(* CODESYS project xlh_gantry_00_04.project
   Description: Receives some incoming messages and echoes them with CAN-ID +1
   Company: 3S - Smart Software Solutions GmbH
   Version: 1.0.0.0
   Title: CAN Bus API Example
   Author: 3S - Smart Software Solutions GmbH

Project tree, tasks and I/O mapping:
  xLH_base : CODESYS Control for Raspberry Pi 64 SL, CODESYS, order no. 2302000009, version 4.20.0.0
    application app
      libraries: Standard, 3.5.22.0 (System); Util, 3.5.22.0 (System); VisuDialogs, * (System); Memory, * (3S - Smart Software Solutions GmbH); CmpBitmapPool, * (System); CAN API, 1.0.0.4 (CODESYS); MemoryUtils, * (3S - Smart Software Solutions GmbH); CAA CiA 405, 4.3.0.0 (CODESYS)
      task CANOPEN_TASK (cyclic, interval 1 ms, priority 1) calls nothing
      task VISU_TASK (cyclic, interval 100 ms, priority 31) calls VisuElems.Visu_Prg
      task MAIN_TASK (cyclic, interval 4 ms, priority 2) calls io, MAIN_CALLER
      task SoftMotion_PlanningTask (cyclic, interval t#2ms, priority 15) calls nothing
      program MAIN_CALLER [ST]
      trace Trace_AxX (task MAIN_TASK): x_axis.fActPosition, x_axis.fSetPosition, x_axis.fSetAcceleration, x_axis.fActAcceleration, x_axis.fSetVelocity, x_axis.fActVelocity, io.motion.adiFrequency[1]
      visualisation Visualization
      trace Trace (task MAIN_TASK): MC.diPosition, MC.iSetSpeed, MC.iDebug2Pos, MC.iDebug1Mileage, MC.auiUltrasonic[1], MC.fbReadStatusLoopTime.udiValue, MC.iSpeed2, MC.iSpeed1, MC.iPitch
      data type MOTION_CONTROL_BYTE
      MOTION_BASE/
        function block FB_XLH_MOTION_AXIS_SIMPLE_ES [ST]: mRead
        function block FB_PLC_OPEN_AXIS [ST]: plcOpen, executeToFalse
        function block FB_XLH_MOTION_AXIS_SIMPLE [ST]
        function block FB_XLH_MOTION_AXIS_BASE [ST]: mRead, mWrite
        function block FB_AXG_MOVE_ABSOLUTE [ST]
        function block FB_AXG_MOVE_RELATIVE [ST]
        function block FB_AXG_PICK_AND_PLACE [ST]
        function block FB_KALMAN_FILTER [ST]: reset
      IO/
        function block FB_XLH_MOTION [ST]: read, write
        program io [ST]: read, write
        function block FB_XLH_GPIO [ST]: read, write
        function block FB_XLH_DXL_RGB [ST]: read, write
      program MC [ST]: write, read, axSmExecuteToFalse, axGexecuteToFalse
      axis group AxisGroup: TRAFO.Kin_Gantry3, axes x_axis, y_axis, z_axis
      trace Trace_AxZ (task MAIN_TASK): z_axis.fActPosition, z_axis.fSetPosition, z_axis.fSetAcceleration, z_axis.fActAcceleration, z_axis.fSetVelocity, z_axis.fActVelocity, io.motion.adiFrequency[3]
    CANbus : CANbus, CODESYS, version 4.3.0.0
        settings: Baudrate = 1000 kbit/s
      CANopen_Manager : CANopen_Manager, CODESYS, version 4.3.0.0
          settings: NMT Start All = TRUE; Polling of optional slaves = FALSE; ConfigVersion = 50659584
        xlh_dynamixel_rgb : xlh_stamp_dynamixel_rgb, xemax ag, order no. 0, version Revision=16#00000001, FileVersion=1.0 (disabled)
            settings: NODEIDSAVED = 2; SDO Timeout = 1000000; PDO_Autoconfig = FALSE; EXPERTSETTINGS = FALSE; PDO 16#1400.COBID = 16#00000202; Process by CANopenManager = TRUE; PDO 16#1401.COBID = 16#00000302; Process by CANopenManager = TRUE; PDO 16#1402.COBID = 16#00000402; Process by CANopenManager = TRUE; PDO 16#1800.COBID = 16#00000182; Process by CANopenManager = TRUE; Dxl 1 Control.Subindex = 16#01; Dxl 1 Position.Subindex = 16#02; Dxl 1 Velocity.Subindex = 16#03; Dxl 2 Control.Subindex = 16#04; Dxl 2 Position.Subindex = 16#05; Dxl 2 Velocity.Subindex = 16#06; RGB red.Subindex = 16#01; RGB green.Subindex = 16#02; RGB blue.Subindex = 16#03; Dxl 1  Position read.Subindex = 16#01; Dxl 1 Current read.Subindex = 16#02; Dxl 2  Position read.Subindex = 16#03; Dxl 2 Current read.Subindex = 16#04; SDO List.Set COB-ID sync.Index = 16#1005; SDO List.Set COB-ID sync.Subindex = 16#00; SDO List.Set COB-ID sync.Value = 16#00000080; SDO List.Set COB-ID sync.Size = 32; SDO List.Set COB-ID sync.AbortIfError = FALSE; SDO List.Set COB-ID sync.JumpToLine = FALSE; SDO List.Set COB-ID sync.Line = 0; SDO List.Set communication cycle period.Index = 16#1006; SDO List.Set communication cycle period.Subindex = 16#00; SDO List.Set communication cycle period.Value = 16#00000000; SDO List.Set communication cycle period.Size = 32; SDO List.Set communication cycle period.AbortIfError = FALSE; SDO List.Set communication cycle period.JumpToLine = FALSE; SDO List.Set communication cycle period.Line = 0; SDO List.Set Guardtime.Index = 16#100C;
              SDO List.Set Guardtime.Subindex = 16#00; SDO List.Set Guardtime.Value = 16#000000C8; SDO List.Set Guardtime.Size = 16; SDO List.Set Guardtime.AbortIfError = FALSE; SDO List.Set Guardtime.JumpToLine = FALSE; SDO List.Set Guardtime.Line = 0; SDO List.Set Lifetime.Index = 16#100D; SDO List.Set Lifetime.Subindex = 16#00; SDO List.Set Lifetime.Value = 16#00000003; SDO List.Set Lifetime.Size = 8; SDO List.Set Lifetime.AbortIfError = FALSE; SDO List.Set Lifetime.JumpToLine = FALSE; SDO List.Set Lifetime.Line = 0; SDO List.Set Heartbeat Consumer.Index = 16#1016; SDO List.Set Heartbeat Consumer.Subindex = 16#01; SDO List.Set Heartbeat Consumer.Value = 0; SDO List.Set Heartbeat Consumer.Size = 32; SDO List.Set Heartbeat Consumer.AbortIfError = FALSE; SDO List.Set Heartbeat Consumer.JumpToLine = FALSE; SDO List.Set Heartbeat Consumer.Line = 0; SDO List.Disable PDO.Index = 16#1400; SDO List.Disable PDO.Subindex = 16#01; SDO List.Disable PDO.Value = 16#80000202; SDO List.Disable PDO.Size = 32; SDO List.Disable PDO.AbortIfError = FALSE; SDO List.Disable PDO.JumpToLine = FALSE; SDO List.Disable PDO.Line = 0; SDO List.Set transmission type.Index = 16#1400; SDO List.Set transmission type.Subindex = 16#02; SDO List.Set transmission type.Value = 16#FF; SDO List.Set transmission type.Size = 8; SDO List.Set transmission type.AbortIfError = FALSE; SDO List.Set transmission type.JumpToLine = FALSE; SDO List.Set transmission type.Line = 0; SDO List.Set and enable COB-ID.Index = 16#1400; SDO List.Set and enable COB-ID.Subindex = 16#01; SDO List.Set and enable COB-ID.Value = 16#00000202; SDO List.Set and enable COB-ID.Size = 32; SDO List.Set and enable COB-ID.AbortIfError = FALSE; SDO List.Set and enable COB-ID.JumpToLine = FALSE;
              SDO List.Set and enable COB-ID.Line = 0; SDO List.Disable PDO.Index = 16#1401; SDO List.Disable PDO.Subindex = 16#01; SDO List.Disable PDO.Value = 16#80000302; SDO List.Disable PDO.Size = 32; SDO List.Disable PDO.AbortIfError = FALSE; SDO List.Disable PDO.JumpToLine = FALSE; SDO List.Disable PDO.Line = 0; SDO List.Set transmission type.Index = 16#1401; SDO List.Set transmission type.Subindex = 16#02; SDO List.Set transmission type.Value = 16#FF; SDO List.Set transmission type.Size = 8; SDO List.Set transmission type.AbortIfError = FALSE; SDO List.Set transmission type.JumpToLine = FALSE; SDO List.Set transmission type.Line = 0; SDO List.Set and enable COB-ID.Index = 16#1401; SDO List.Set and enable COB-ID.Subindex = 16#01; SDO List.Set and enable COB-ID.Value = 16#00000302; SDO List.Set and enable COB-ID.Size = 32; SDO List.Set and enable COB-ID.AbortIfError = FALSE; SDO List.Set and enable COB-ID.JumpToLine = FALSE; SDO List.Set and enable COB-ID.Line = 0; SDO List.Disable PDO.Index = 16#1402; SDO List.Disable PDO.Subindex = 16#01; SDO List.Disable PDO.Value = 16#80000402; SDO List.Disable PDO.Size = 32; SDO List.Disable PDO.AbortIfError = FALSE; SDO List.Disable PDO.JumpToLine = FALSE; SDO List.Disable PDO.Line = 0; SDO List.Set transmission type.Index = 16#1402; SDO List.Set transmission type.Subindex = 16#02; SDO List.Set transmission type.Value = 16#FF; SDO List.Set transmission type.Size = 8; SDO List.Set transmission type.AbortIfError = FALSE; SDO List.Set transmission type.JumpToLine = FALSE; SDO List.Set transmission type.Line = 0; SDO List.Set and enable COB-ID.Index = 16#1402; SDO List.Set and enable COB-ID.Subindex = 16#01; SDO List.Set and enable COB-ID.Value = 16#00000402; SDO List.Set and enable COB-ID.Size = 32;
              SDO List.Set and enable COB-ID.AbortIfError = FALSE; SDO List.Set and enable COB-ID.JumpToLine = FALSE; SDO List.Set and enable COB-ID.Line = 0; SDO List.Disable PDO.Index = 16#1800; SDO List.Disable PDO.Subindex = 16#01; SDO List.Disable PDO.Value = 16#80000182; SDO List.Disable PDO.Size = 32; SDO List.Disable PDO.AbortIfError = FALSE; SDO List.Disable PDO.JumpToLine = FALSE; SDO List.Disable PDO.Line = 0; SDO List.Set transmission type.Index = 16#1800; SDO List.Set transmission type.Subindex = 16#02; SDO List.Set transmission type.Value = 16#FF; SDO List.Set transmission type.Size = 8; SDO List.Set transmission type.AbortIfError = FALSE; SDO List.Set transmission type.JumpToLine = FALSE; SDO List.Set transmission type.Line = 0; SDO List.Set inhibit time.Index = 16#1800; SDO List.Set inhibit time.Subindex = 16#03; SDO List.Set inhibit time.Value = 16#0000; SDO List.Set inhibit time.Size = 16; SDO List.Set inhibit time.AbortIfError = FALSE; SDO List.Set inhibit time.JumpToLine = FALSE; SDO List.Set inhibit time.Line = 0; SDO List.Set event time.Index = 16#1800; SDO List.Set event time.Subindex = 16#05; SDO List.Set event time.Value = 16#0000; SDO List.Set event time.Size = 16; SDO List.Set event time.AbortIfError = FALSE; SDO List.Set event time.JumpToLine = FALSE; SDO List.Set event time.Line = 0; SDO List.Set and enable COB-ID.Index = 16#1800; SDO List.Set and enable COB-ID.Subindex = 16#01; SDO List.Set and enable COB-ID.Value = 16#00000182; SDO List.Set and enable COB-ID.Size = 32; SDO List.Set and enable COB-ID.AbortIfError = FALSE; SDO List.Set and enable COB-ID.JumpToLine = FALSE; SDO List.Set and enable COB-ID.Line = 0; ConfigVersion = 50659584
            output app.io.dxlRgb.bDxl1Torque : BOOL  // Dxl 1 Control.Bit0
            output app.io.dxlRgb.bDxl1Led : BOOL  // Dxl 1 Control.Bit1
            output app.io.dxlRgb.uiDxl1Position : UINT  // Dxl 1 Position
            output app.io.dxlRgb.uiDxl1Velocity : UINT  // Dxl 1 Velocity
            output app.io.dxlRgb.bDxl2Torque : BOOL  // Dxl 2 Control.Bit0
            output app.io.dxlRgb.bDxl2Led : BOOL  // Dxl 2 Control.Bit1
            output app.io.dxlRgb.uiDxl2Position : UINT  // Dxl 2 Position
            output app.io.dxlRgb.uiDxl2Velocity : UINT  // Dxl 2 Velocity
            output app.io.dxlRgb.byRgbRed : USINT  // RGB red
            output app.io.dxlRgb.byRgbGreen : USINT  // RGB green
            output app.io.dxlRgb.byRgbBlue : USINT  // RGB blue
            input  app.io.dxlRgb.uiDxl1PositionGet : UINT  // Dxl 1  Position read
            input  app.io.dxlRgb.iDxl1CurrentGet : INT  // Dxl 1 Current read
            input  app.io.dxlRgb.uiDxl2PositionGet : UINT  // Dxl 2  Position read
            input  app.io.dxlRgb.iDxl2CurrentGet : INT  // Dxl 2 Current read
            unmapped channels: Dxl 1 Control, Dxl 2 Control
        xlh_motion : xlh_motion, xemax ag, order no. 0, version Revision=16#00000001, FileVersion=1.0
            settings: NODEIDSAVED = 1; SDO Timeout = 1000000; PDO_Autoconfig = FALSE; EXPERTSETTINGS = True; PDO 16#1400.COBID = 16#00000201; Process by CANopenManager = TRUE; PDO 16#1401.COBID = 16#00000301; Process by CANopenManager = TRUE; PDO 16#1402.COBID = 16#00000401; Process by CANopenManager = TRUE; PDO 16#1403.COBID = 16#00000501; Process by CANopenManager = TRUE; PDO 16#1800.COBID = 16#00000181; Process by CANopenManager = TRUE; PDO 16#1801.COBID = 16#00000281; Process by CANopenManager = TRUE; PDO 16#1802.COBID = 16#00000381; Process by CANopenManager = TRUE; Control 1.Subindex = 16#01; Control 2.Subindex = 16#02; Control 3.Subindex = 16#03; Control 4.Subindex = 16#04; Outputs 0-7.Subindex = 16#01; Outputs 8-15.Subindex = 16#02; Magnet Duty Cycle.Subindex = 16#01; Freqeuncy 1.Subindex = 16#05; Freqeuncy 2.Subindex = 16#06; Freqeuncy 3.Subindex = 16#07; Freqeuncy 4.Subindex = 16#08; Servo 1.Subindex = 16#01; Servo 2.Subindex = 16#02; Servo 3.Subindex = 16#03; Servo 4.Subindex = 16#04; Servo 5.Subindex = 16#05; Servo 6.Subindex = 16#06; Servo 7.Subindex = 16#07; Servo 8.Subindex = 16#08; Position 1.Subindex = 16#01; Position 2.Subindex = 16#02; Position 3.Subindex = 16#03;
              Position 4.Subindex = 16#04; Inputs 0-7.Subindex = 16#01; Inputs 8-15.Subindex = 16#02; Inputs CLK.Subindex = 16#03; SDO List.Set COB-ID sync.Index = 16#1005; SDO List.Set COB-ID sync.Subindex = 16#00; SDO List.Set COB-ID sync.Value = 16#00000080; SDO List.Set COB-ID sync.Size = 32; SDO List.Set COB-ID sync.AbortIfError = FALSE; SDO List.Set COB-ID sync.JumpToLine = FALSE; SDO List.Set COB-ID sync.Line = 0; SDO List.Set communication cycle period.Index = 16#1006; SDO List.Set communication cycle period.Subindex = 16#00; SDO List.Set communication cycle period.Value = 16#00000000; SDO List.Set communication cycle period.Size = 32; SDO List.Set communication cycle period.AbortIfError = FALSE; SDO List.Set communication cycle period.JumpToLine = FALSE; SDO List.Set communication cycle period.Line = 0; SDO List.Set Guardtime.Index = 16#100C; SDO List.Set Guardtime.Subindex = 16#00; SDO List.Set Guardtime.Value = 16#000000C8; SDO List.Set Guardtime.Size = 16; SDO List.Set Guardtime.AbortIfError = FALSE; SDO List.Set Guardtime.JumpToLine = FALSE; SDO List.Set Guardtime.Line = 0; SDO List.Set Lifetime.Index = 16#100D; SDO List.Set Lifetime.Subindex = 16#00; SDO List.Set Lifetime.Value = 16#00000003; SDO List.Set Lifetime.Size = 8; SDO List.Set Lifetime.AbortIfError = FALSE; SDO List.Set Lifetime.JumpToLine = FALSE; SDO List.Set Lifetime.Line = 0; SDO List.Set Heartbeat Consumer.Index = 16#1016; SDO List.Set Heartbeat Consumer.Subindex = 16#01; SDO List.Set Heartbeat Consumer.Value = 0; SDO List.Set Heartbeat Consumer.Size = 32; SDO List.Set Heartbeat Consumer.AbortIfError = FALSE; SDO List.Set Heartbeat Consumer.JumpToLine = FALSE; SDO List.Set Heartbeat Consumer.Line = 0; SDO List.Disable PDO.Index = 16#1400;
              SDO List.Disable PDO.Subindex = 16#01; SDO List.Disable PDO.Value = 16#80000201; SDO List.Disable PDO.Size = 32; SDO List.Disable PDO.AbortIfError = FALSE; SDO List.Disable PDO.JumpToLine = FALSE; SDO List.Disable PDO.Line = 0; SDO List.Set transmission type.Index = 16#1400; SDO List.Set transmission type.Subindex = 16#02; SDO List.Set transmission type.Value = 16#FF; SDO List.Set transmission type.Size = 8; SDO List.Set transmission type.AbortIfError = FALSE; SDO List.Set transmission type.JumpToLine = FALSE; SDO List.Set transmission type.Line = 0; SDO List.Set and enable COB-ID.Index = 16#1400; SDO List.Set and enable COB-ID.Subindex = 16#01; SDO List.Set and enable COB-ID.Value = 16#00000201; SDO List.Set and enable COB-ID.Size = 32; SDO List.Set and enable COB-ID.AbortIfError = FALSE; SDO List.Set and enable COB-ID.JumpToLine = FALSE; SDO List.Set and enable COB-ID.Line = 0; SDO List.Disable PDO.Index = 16#1401; SDO List.Disable PDO.Subindex = 16#01; SDO List.Disable PDO.Value = 16#80000301; SDO List.Disable PDO.Size = 32; SDO List.Disable PDO.AbortIfError = FALSE; SDO List.Disable PDO.JumpToLine = FALSE; SDO List.Disable PDO.Line = 0; SDO List.Set transmission type.Index = 16#1401; SDO List.Set transmission type.Subindex = 16#02; SDO List.Set transmission type.Value = 16#FF; SDO List.Set transmission type.Size = 8; SDO List.Set transmission type.AbortIfError = FALSE; SDO List.Set transmission type.JumpToLine = FALSE; SDO List.Set transmission type.Line = 0; SDO List.Set and enable COB-ID.Index = 16#1401; SDO List.Set and enable COB-ID.Subindex = 16#01; SDO List.Set and enable COB-ID.Value = 16#00000301; SDO List.Set and enable COB-ID.Size = 32; SDO List.Set and enable COB-ID.AbortIfError = FALSE; SDO List.Set and enable COB-ID.JumpToLine = FALSE;
              SDO List.Set and enable COB-ID.Line = 0; SDO List.Disable PDO.Index = 16#1402; SDO List.Disable PDO.Subindex = 16#01; SDO List.Disable PDO.Value = 16#80000401; SDO List.Disable PDO.Size = 32; SDO List.Disable PDO.AbortIfError = FALSE; SDO List.Disable PDO.JumpToLine = FALSE; SDO List.Disable PDO.Line = 0; SDO List.Set transmission type.Index = 16#1402; SDO List.Set transmission type.Subindex = 16#02; SDO List.Set transmission type.Value = 16#FF; SDO List.Set transmission type.Size = 8; SDO List.Set transmission type.AbortIfError = FALSE; SDO List.Set transmission type.JumpToLine = FALSE; SDO List.Set transmission type.Line = 0; SDO List.Set and enable COB-ID.Index = 16#1402; SDO List.Set and enable COB-ID.Subindex = 16#01; SDO List.Set and enable COB-ID.Value = 16#00000401; SDO List.Set and enable COB-ID.Size = 32; SDO List.Set and enable COB-ID.AbortIfError = FALSE; SDO List.Set and enable COB-ID.JumpToLine = FALSE; SDO List.Set and enable COB-ID.Line = 0; SDO List.Disable PDO.Index = 16#1403; SDO List.Disable PDO.Subindex = 16#01; SDO List.Disable PDO.Value = 16#80000501; SDO List.Disable PDO.Size = 32; SDO List.Disable PDO.AbortIfError = FALSE; SDO List.Disable PDO.JumpToLine = FALSE; SDO List.Disable PDO.Line = 0; SDO List.Set transmission type.Index = 16#1403; SDO List.Set transmission type.Subindex = 16#02; SDO List.Set transmission type.Value = 16#FF; SDO List.Set transmission type.Size = 8; SDO List.Set transmission type.AbortIfError = FALSE; SDO List.Set transmission type.JumpToLine = FALSE; SDO List.Set transmission type.Line = 0; SDO List.Set and enable COB-ID.Index = 16#1403; SDO List.Set and enable COB-ID.Subindex = 16#01; SDO List.Set and enable COB-ID.Value = 16#00000501; SDO List.Set and enable COB-ID.Size = 32;
              SDO List.Set and enable COB-ID.AbortIfError = FALSE; SDO List.Set and enable COB-ID.JumpToLine = FALSE; SDO List.Set and enable COB-ID.Line = 0; SDO List.Disable PDO.Index = 16#1800; SDO List.Disable PDO.Subindex = 16#01; SDO List.Disable PDO.Value = 16#80000181; SDO List.Disable PDO.Size = 32; SDO List.Disable PDO.AbortIfError = FALSE; SDO List.Disable PDO.JumpToLine = FALSE; SDO List.Disable PDO.Line = 0; SDO List.Set transmission type.Index = 16#1800; SDO List.Set transmission type.Subindex = 16#02; SDO List.Set transmission type.Value = 16#FF; SDO List.Set transmission type.Size = 8; SDO List.Set transmission type.AbortIfError = FALSE; SDO List.Set transmission type.JumpToLine = FALSE; SDO List.Set transmission type.Line = 0; SDO List.Set inhibit time.Index = 16#1800; SDO List.Set inhibit time.Subindex = 16#03; SDO List.Set inhibit time.Value = 16#0000; SDO List.Set inhibit time.Size = 16; SDO List.Set inhibit time.AbortIfError = FALSE; SDO List.Set inhibit time.JumpToLine = FALSE; SDO List.Set inhibit time.Line = 0; SDO List.Set event time.Index = 16#1800; SDO List.Set event time.Subindex = 16#05; SDO List.Set event time.Value = 16#0000; SDO List.Set event time.Size = 16; SDO List.Set event time.AbortIfError = FALSE; SDO List.Set event time.JumpToLine = FALSE; SDO List.Set event time.Line = 0; SDO List.Set and enable COB-ID.Index = 16#1800; SDO List.Set and enable COB-ID.Subindex = 16#01; SDO List.Set and enable COB-ID.Value = 16#00000181; SDO List.Set and enable COB-ID.Size = 32; SDO List.Set and enable COB-ID.AbortIfError = FALSE; SDO List.Set and enable COB-ID.JumpToLine = FALSE; SDO List.Set and enable COB-ID.Line = 0; SDO List.Disable PDO.Index = 16#1801; SDO List.Disable PDO.Subindex = 16#01;
              SDO List.Disable PDO.Value = 16#80000281; SDO List.Disable PDO.Size = 32; SDO List.Disable PDO.AbortIfError = FALSE; SDO List.Disable PDO.JumpToLine = FALSE; SDO List.Disable PDO.Line = 0; SDO List.Set transmission type.Index = 16#1801; SDO List.Set transmission type.Subindex = 16#02; SDO List.Set transmission type.Value = 16#FF; SDO List.Set transmission type.Size = 8; SDO List.Set transmission type.AbortIfError = FALSE; SDO List.Set transmission type.JumpToLine = FALSE; SDO List.Set transmission type.Line = 0; SDO List.Set inhibit time.Index = 16#1801; SDO List.Set inhibit time.Subindex = 16#03; SDO List.Set inhibit time.Value = 16#0000; SDO List.Set inhibit time.Size = 16; SDO List.Set inhibit time.AbortIfError = FALSE; SDO List.Set inhibit time.JumpToLine = FALSE; SDO List.Set inhibit time.Line = 0; SDO List.Set event time.Index = 16#1801; SDO List.Set event time.Subindex = 16#05; SDO List.Set event time.Value = 16#0000; SDO List.Set event time.Size = 16; SDO List.Set event time.AbortIfError = FALSE; SDO List.Set event time.JumpToLine = FALSE; SDO List.Set event time.Line = 0; SDO List.Set and enable COB-ID.Index = 16#1801; SDO List.Set and enable COB-ID.Subindex = 16#01; SDO List.Set and enable COB-ID.Value = 16#00000281; SDO List.Set and enable COB-ID.Size = 32; SDO List.Set and enable COB-ID.AbortIfError = FALSE; SDO List.Set and enable COB-ID.JumpToLine = FALSE; SDO List.Set and enable COB-ID.Line = 0; SDO List.Disable PDO.Index = 16#1802; SDO List.Disable PDO.Subindex = 16#01; SDO List.Disable PDO.Value = 16#80000381; SDO List.Disable PDO.Size = 32; SDO List.Disable PDO.AbortIfError = FALSE; SDO List.Disable PDO.JumpToLine = FALSE; SDO List.Disable PDO.Line = 0;
              SDO List.Set transmission type.Index = 16#1802; SDO List.Set transmission type.Subindex = 16#02; SDO List.Set transmission type.Value = 16#FF; SDO List.Set transmission type.Size = 8; SDO List.Set transmission type.AbortIfError = FALSE; SDO List.Set transmission type.JumpToLine = FALSE; SDO List.Set transmission type.Line = 0; SDO List.Set inhibit time.Index = 16#1802; SDO List.Set inhibit time.Subindex = 16#03; SDO List.Set inhibit time.Value = 16#0000; SDO List.Set inhibit time.Size = 16; SDO List.Set inhibit time.AbortIfError = FALSE; SDO List.Set inhibit time.JumpToLine = FALSE; SDO List.Set inhibit time.Line = 0; SDO List.Set event time.Index = 16#1802; SDO List.Set event time.Subindex = 16#05; SDO List.Set event time.Value = 16#0000; SDO List.Set event time.Size = 16; SDO List.Set event time.AbortIfError = FALSE; SDO List.Set event time.JumpToLine = FALSE; SDO List.Set event time.Line = 0; SDO List.Set and enable COB-ID.Index = 16#1802; SDO List.Set and enable COB-ID.Subindex = 16#01; SDO List.Set and enable COB-ID.Value = 16#00000381; SDO List.Set and enable COB-ID.Size = 32; SDO List.Set and enable COB-ID.AbortIfError = FALSE; SDO List.Set and enable COB-ID.JumpToLine = FALSE; SDO List.Set and enable COB-ID.Line = 0; ConfigVersion = 50659584
            output app.io.motion.abyControl[1] : USINT  // Control 1
            output app.io.motion.abyControl[2] : USINT  // Control 2
            output app.io.motion.abyControl[3] : USINT  // Control 3
            output app.io.motion.abyControl[4] : USINT  // Control 4
            output app.io.motion.abyOutputs[1] : USINT  // Outputs 0-7
            output app.io.motion.abyOutputs[2] : USINT  // Outputs 8-15
            output app.io.motion.uiMagnetDutyCycle : UINT  // Magnet Duty Cycle
            output app.io.motion.adiFrequency[1] : DINT  // Freqeuncy 1
            output app.io.motion.adiFrequency[2] : DINT  // Freqeuncy 2
            output app.io.motion.adiFrequency[3] : DINT  // Freqeuncy 3
            output app.io.motion.adiFrequency[4] : DINT  // Freqeuncy 4
            output app.io.motion.ausServo[1] : USINT  // Servo 1
            output app.io.motion.ausServo[2] : USINT  // Servo 2
            output app.io.motion.ausServo[3] : USINT  // Servo 3
            output app.io.motion.ausServo[4] : USINT  // Servo 4
            output app.io.motion.ausServo[5] : USINT  // Servo 5
            output app.io.motion.ausServo[6] : USINT  // Servo 6
            output app.io.motion.ausServo[7] : USINT  // Servo 7
            output app.io.motion.ausServo[8] : USINT  // Servo 8
            input  app.io.motion.adiPosition[1] : DINT  // Position 1
            input  app.io.motion.adiPosition[2] : DINT  // Position 2
            input  app.io.motion.adiPosition[3] : DINT  // Position 3
            input  app.io.motion.adiPosition[4] : DINT  // Position 4
            input  app.io.motion.abyInputs[1] : USINT  // Inputs 0-7
            input  app.io.motion.bAxXsw : BOOL  // Inputs 0-7.Bit0
            input  app.io.motion.bAxYsw : BOOL  // Inputs 0-7.Bit1
            input  app.io.motion.bAxZsw : BOOL  // Inputs 0-7.Bit2
            input  app.io.motion.bSensor : BOOL  // Inputs 0-7.Bit3
            input  app.io.motion.abyInputs[2] : USINT  // Inputs 8-15
            input  app.io.motion.abyInputs[3] : USINT  // Inputs CLK
    Camera device
      <Leer>
    GPIOs_A_B : GPIOs B+/Pi2, CODESYS, version 4.20.0.0
        input  app.io.gpio.bSw1 : BOOL  // digital inputs (GPIO0..GPIO31).Bit4
        input  app.io.gpio.bSw2 : BOOL  // digital inputs (GPIO0..GPIO31).Bit5
        input  app.io.gpio.bSw3 : BOOL  // digital inputs (GPIO0..GPIO31).Bit6
        input  app.io.gpio.bSw4 : BOOL  // digital inputs (GPIO0..GPIO31).Bit12
        input  app.io.gpio.bSw5 : BOOL  // digital inputs (GPIO0..GPIO31).Bit13
        input  app.io.gpio.bSw6 : BOOL  // digital inputs (GPIO0..GPIO31).Bit16
        input  app.io.gpio.bSw7 : BOOL  // digital inputs (GPIO0..GPIO31).Bit17
        input  app.io.gpio.bSw8 : BOOL  // digital inputs (GPIO0..GPIO31).Bit19
        output app.io.gpio.bLed1 : BOOL  // digital outputs (GPIO0..GPIO31).Bit20
        output app.io.gpio.bLed2 : BOOL  // digital outputs (GPIO0..GPIO31).Bit21
        output app.io.gpio.bLed3 : BOOL  // digital outputs (GPIO0..GPIO31).Bit22
        output app.io.gpio.bLed4 : BOOL  // digital outputs (GPIO0..GPIO31).Bit23
        output app.io.gpio.bLed5 : BOOL  // digital outputs (GPIO0..GPIO31).Bit24
        output app.io.gpio.bLed6 : BOOL  // digital outputs (GPIO0..GPIO31).Bit26
        output app.io.gpio.bLed7 : BOOL  // digital outputs (GPIO0..GPIO31).Bit27
        unmapped channels: digital inputs (GPIO0..GPIO31), digital outputs (GPIO0..GPIO31)
    I²C
    SoftMotion General Axis Pool
      x_axis : SM_Drive_PosControl, CODESYS, order no. 1805, version 4.18.0.0
          settings: wDriveID = 0; dwRatioTechUnitsDenom = 101846; iRatioTechUnitsNum = 125; eRampType = 0; fSWMaxVelocity = 50; fSWMaxAcceleration = 100; fSWMaxDeceleration = 100; fSWMaxJerk = 1000; fSWLimitNegative = -1000; ScalingIncs = 814768; ScalingUnits = 1000; IsLinearMotor = TRUE; MaximumOutputVelocityInt = 40738; MinimumOutputVelocityInt = -40738; Kp = 0.005; MaxFollowingError = 1; PartVelocityPilotControl = 1; DeadTime = 1
      z_axis : SM_Drive_PosControl, CODESYS, order no. 1805, version 4.18.0.0
          settings: wDriveID = 2; dwRatioTechUnitsDenom = 101846; iRatioTechUnitsNum = -125; eRampType = 0; fSWMaxVelocity = 50; fSWMaxAcceleration = 100; fSWMaxDeceleration = 100; fSWMaxJerk = 1000; fSWLimitNegative = -1000; ScalingIncs = 814768; ScalingUnits = 1000; InvertDirection = TRUE; IsLinearMotor = TRUE; MaximumOutputVelocityInt = 40738; MinimumOutputVelocityInt = -40738; Kp = 0.005; MaxFollowingError = 1; DeadTime = 1
      y_axis : SM_Drive_PosControl, CODESYS, order no. 1805, version 4.18.0.0
          settings: dwRatioTechUnitsDenom = 101846; iRatioTechUnitsNum = -125; eRampType = 0; fSWMaxVelocity = 50; fSWMaxAcceleration = 100; fSWMaxDeceleration = 100; fSWMaxJerk = 1000; fSWLimitNegative = -1000; ScalingIncs = 814768; ScalingUnits = 1000; InvertDirection = TRUE; IsLinearMotor = TRUE; MaximumOutputVelocityInt = 40738; MinimumOutputVelocityInt = -40738; Kp = 0.005; MaxFollowingError = 1; PartVelocityPilotControl = 1; DeadTime = 1
      a_axis : SM_Drive_PosControl, CODESYS, order no. 1805, version 4.18.0.0
          settings: wDriveID = 3; dwRatioTechUnitsDenom = 101846; iRatioTechUnitsNum = -125; eRampType = 0; fSWMaxVelocity = 50; fSWMaxAcceleration = 100; fSWMaxDeceleration = 100; fSWMaxJerk = 1000; fSWLimitNegative = -1000.0; ScalingIncs = 814768; ScalingUnits = 1000; InvertDirection = TRUE; IsLinearMotor = TRUE; MaximumOutputVelocityInt = 40738; MinimumOutputVelocityInt = -40738; Kp = 0.005; MaxFollowingError = 1; DeadTime = 1
    Onewire
    SPI
  libraries: VisuSymbols, 4.5.0.0 (System); DepictorBase, 1.2.0.0 (CODESYS)
  text list GlobalTextList
  5ce3da45-db07-42e7-a21c-a00fff4ed8f6|C:\Users\phe\Downloads\Musterloesung_FUP.PNG
*)

// xLH_base/app/MOTION_CONTROL_BYTE
TYPE MOTION_CONTROL_BYTE :
STRUCT
	bEnable: BOOL;
	bDir: BOOL;
	bReset: BOOL;
	bInverted: BOOL;
	bInMotion: BOOL;
	bMoveWithoutPulse: BOOL;
END_STRUCT
END_TYPE

// xLH_base/app/IO/io
PROGRAM io 
VAR_INPUT
	gpio: FB_XLH_GPIO;	
	dxlRgb: FB_XLH_DXL_RGB;
	motion: FB_XLH_MOTION;
	bMagnet: bool;
	

	fbXlhMotionAxisX: FB_XLH_MOTION_AXIS_SIMPLE_ES;
	fbXlhMotionAxisY: FB_XLH_MOTION_AXIS_SIMPLE_ES;
	fbXlhMotionAxisZ: FB_XLH_MOTION_AXIS_SIMPLE_ES;
	fbXlhMotionAxisA: FB_XLH_MOTION_AXIS_SIMPLE;
END_VAR
VAR	
	bStartup: BOOL := TRUE;

	bDummy: BOOL;
	byDummy: BYTE;
	usDummy: USINT;
	iDummy: INT;
	uiDummy: UINT;
	diDummy: DINT;
	udiDummy: UDINT;
	rDummy: REAL;
	fDummy: LREAL;
END_VAR

IF bStartup THEN
	bStartup := FALSE;
	io.dxlRgb.bDxl1Torque := TRUE;
	io.dxlRgb.uiDxl1Position := 1024;
	io.dxlRgb.uiDxl1Velocity := 50;
	
	io.dxlRgb.bDxl2Torque := TRUE;
	io.dxlRgb.uiDxl2Position := 1024;
	io.dxlRgb.uiDxl2Velocity := 50;
	
	io.dxlRgb.byRgbRed := 0;
	io.dxlRgb.byRgbGreen := 0;
	io.dxlRgb.byRgbBlue := 0;
	
	io.motion.ausServo[1] := 128;
	
	fbXlhMotionAxisX.pfbAxisPlcOpen := ADR(MC.axX);
	fbXlhMotionAxisX.pAxis := ADR(x_axis);
	fbXlhMotionAxisX.pbEs := ADR(io.motion.bAxXsw);
	
	fbXlhMotionAxisY.pfbAxisPlcOpen := ADR(MC.axY);
	fbXlhMotionAxisY.pAxis := ADR(y_axis);
	fbXlhMotionAxisY.pbEs := ADR(io.motion.bAxYsw);

	fbXlhMotionAxisZ.pfbAxisPlcOpen := ADR(MC.axZ);
	fbXlhMotionAxisZ.pAxis := ADR(z_axis);
	fbXlhMotionAxisZ.pbEs := ADR(io.motion.bAxZsw);
	
	fbXlhMotionAxisA.pfbAxisPlcOpen := ADR(MC.axA);
	fbXlhMotionAxisA.pAxis := ADR(a_axis);
	//fbXlhMotionAxisA.pbEs := ADR(bAxAsw);
	
	
	motion.pfbXlhMotionAxis[1] := ADR(fbXlhMotionAxisX);
	motion.pfbXlhMotionAxis[2] := ADR(fbXlhMotionAxisY);
	motion.pfbXlhMotionAxis[3] := ADR(fbXlhMotionAxisZ);
	motion.pfbXlhMotionAxis[4] := ADR(fbXlhMotionAxisA);
END_IF

IF bMagnet THEN
	motion.uiMagnetDutyCycle := 4095;
ELSE
	motion.uiMagnetDutyCycle := 0;
END_IF




byDummy := io.motion.abyInputs[1];
bDummy := io.motion.bSensor;
uiDummy := io.motion.uiMagnetDutyCycle;

fDummy := y_axis.fActPosition;
fDummy := y_axis.fSetPosition;
fDummy := y_axis.fActVelocity;
fDummy := y_axis.fSetVelocity;
fDummy := y_axis.fActAcceleration;
fDummy := y_axis.fSetAcceleration;

usDummy := io.motion.ausServo[1];
io.motion.ausServo[2] := io.motion.ausServo[1];
io.motion.ausServo[3] := io.motion.ausServo[1];
io.motion.ausServo[4] := io.motion.ausServo[1];
io.motion.ausServo[5] := io.motion.ausServo[1];
io.motion.ausServo[6] := io.motion.ausServo[1];
io.motion.ausServo[7] := io.motion.ausServo[1];
io.motion.ausServo[8] := io.motion.ausServo[1];

// Dynamixel + RGB
bDummy := io.dxlRgb.bDxl1Torque;
bDummy := io.dxlRgb.bDxl1Led;
uiDummy := io.dxlRgb.uiDxl1Position;
uiDummy := io.dxlRgb.uiDxl1Velocity;
uiDummy := io.dxlRgb.uiDxl1PositionGet;
iDummy := io.dxlRgb.iDxl1CurrentGet;

bDummy := io.dxlRgb.bDxl2Torque;
bDummy := io.dxlRgb.bDxl2Led;
uiDummy := io.dxlRgb.uiDxl2Position;
uiDummy := io.dxlRgb.uiDxl2Velocity;
uiDummy := io.dxlRgb.uiDxl2PositionGet;
iDummy := io.dxlRgb.iDxl2CurrentGet;

byDummy := io.dxlRgb.byRgbRed;
byDummy := io.dxlRgb.byRgbGreen;
byDummy := io.dxlRgb.byRgbBlue;

METHOD read : BOOL
VAR_INPUT
END_VAR
gpio.read();
dxlRgb.read();
motion.read();
END_METHOD

METHOD write : BOOL
VAR_INPUT
END_VAR
gpio.write();
dxlRgb.write();
motion.write();
END_METHOD

END_PROGRAM

// xLH_base/app/MC
PROGRAM MC
VAR
	iState: INT;	
	
	axX: FB_PLC_OPEN_AXIS := (fVel:=fVEL, fAcc:=fACC_DEC, fDec:=fACC_DEC, fJerk:=fJERK);
	axY: FB_PLC_OPEN_AXIS := (fVel:=fVEL, fAcc:=fACC_DEC, fDec:=fACC_DEC, fJerk:=fJERK);
	axZ: FB_PLC_OPEN_AXIS := (fVel:=fVEL, fAcc:=fACC_DEC, fDec:=fACC_DEC, fJerk:=fJERK);
	axA: FB_PLC_OPEN_AXIS := (fVel:=fVEL, fAcc:=fACC_DEC, fDec:=fACC_DEC, fJerk:=fJERK);	

	//
	baxGenable: BOOL;
	mcAxGenable : MC_GroupEnable;
	mcAxGdisable : MC_GroupDisable;
	mcAxGreset: MC_GroupReset;
	mcAxGsetCoord : MC_SetCoordinateTransform;	
	mcAxGmla: MC_MoveLinearAbsolute := (Velocity := fVEL, Acceleration := fACC_DEC, Deceleration := fACC_DEC, Jerk := fJERK);
	mcAxGmlr: MC_MoveLinearRelative := (Velocity := fVEL, Acceleration := fACC_DEC, Deceleration := fACC_DEC, Jerk := fJERK);	
	mcAxGcoordRef : MC_COORD_REF;
	tPosMC : SMC_POS_REF ;
	grp : SMC_GroupReadSetPosition := (Enable:= TRUE, CoordSystem:= SMC_COORD_SYSTEM.MCS);
	fbAxGmr: FB_AXG_MOVE_RELATIVE;
	fbAxGma: FB_AXG_MOVE_ABSOLUTE;
	fbPickAndPlace: FB_AXG_PICK_AND_PLACE;	
	smcPosRef: SMC_POS_REF;

	//
	bStartup: BOOL := TRUE;
	//
	fbTonDelay1: TON := (PT := TIME#1S0MS);
	fbTonDelay2: TON := (PT := TIME#1S0MS);	
	
	// Aktionsvariablen
	bXp: BOOL;
	bXm: BOOL;
	bYp: BOOL;
	bYm: BOOL;
	bZp: BOOL;
	bZm: BOOL;
	fStep: LREAL := 5.0;
	bAuto: BOOL;
	
	// Testvariablen
	fDistanceTest: LREAL;
	bDummyX: BOOL;
	bDummyY: BOOL;
	bDummyZ: BOOL;
	fDummy: LREAL;
	fPickOffsetX: LREAL;
	fPickOffsetY: LREAL;
	fPlaceOffsetX: LREAL;
	fPlaceOffsetY: LREAL;
	iN: INT;
	fOffsetX: LREAL;
	fOffsetY: LREAL;
	iI: INT;
END_VAR
VAR CONSTANT
	fVEL : LREAL := 30.0;
	fVEL_HOMING : LREAL := 2.0;
    fACC_DEC : LREAL := 20.0;
    fJERK : LREAL := 100.0;	
	
	POS_REF : SMC_POS_REF := (c:= (X:=40.0, Y:=-40.0, Z:=-40.0));
END_VAR

IF bStartup THEN
	bStartup := FALSE;
	axX.pAxis := ADR(x_axis);
	axY.pAxis := ADR(y_axis);
	axZ.pAxis := ADR(z_axis);
	axA.pAxis := ADR(a_axis);	
	
	fbAxGmr.axGmr REF= mcAxGmlr;
	fbAxGmr.axG REF= AxisGroup;  
	fbAxGma.axGma REF= mcAxGmla;
	fbAxGma.axG REF= AxisGroup;

	fbPickAndPlace.fbAxGmr REF= fbAxGmr; 
  	fbPickAndPlace.fbAxGma REF= fbAxGma;
END_IF

MC.read();

// ToDo: Optimierung
mcAxGmla(AxisGroup:= AxisGroup);
mcAxGmlr(AxisGroup:= AxisGroup);
fbAxGmr();
fbAxGma();
fbPickAndPlace();
grp(Enable:=TRUE, AxisGroup:=AxisGroup, Position=>tPosMC);

fDummy := tPosMC.c.X;
fDummy := tPosMC.c.Y;
fDummy := tPosMC.c.Z;
fDummy := tPosMC.c.A;
fDummy := tPosMC.c.B;
fDummy := tPosMC.c.C;

CASE iState OF
	// ============================================================================================
	// STARTUP UND INITIALISIERUNG
	// ============================================================================================
	
	0:		// Startup
		axSmExecuteToFalse();
		axGexecuteToFalse();		
		fbPickAndPlace.bExecute := FALSE;
		bDummyX := TRUE;
		bDummyY := TRUE;
		bDummyZ := TRUE;
		iState := 50;


	50:	// Power der Achsen
		axX.mcp.Enable := TRUE; axX.mcp.bRegulatorOn := TRUE; axX.mcp.bDriveStart := TRUE;
		axY.mcp.Enable := TRUE; axY.mcp.bRegulatorOn := TRUE; axY.mcp.bDriveStart := TRUE;
		axZ.mcp.Enable := TRUE; axZ.mcp.bRegulatorOn := TRUE; axZ.mcp.bDriveStart := TRUE;
		axA.mcp.Enable := TRUE; axA.mcp.bRegulatorOn := TRUE; axA.mcp.bDriveStart := TRUE;
		
		// https://content.helpme-codesys.com/en/libs/SM3_Basic/Current/SM3_Basic/DataTypes/DriveInterface/SMC_AXIS_STATE.html
		IF (axX.mcp.Status AND x_axis.nAxisState = SMC_AXIS_STATE.standstill) AND
		   (axY.mcp.Status AND y_axis.nAxisState = SMC_AXIS_STATE.standstill) AND
		   (axZ.mcp.Status AND z_axis.nAxisState = SMC_AXIS_STATE.standstill) AND
		   (axA.mcp.Status AND a_axis.nAxisState = SMC_AXIS_STATE.standstill) THEN
			MC.axSmExecuteToFalse();
			iState := iState + 10;
		END_IF
		
	60: 
 		iState := 100;

	100:	// Disable der Achsengruppe		
			IF baxGenable THEN
				mcAxGdisable(AxisGroup := AxisGroup, Execute := TRUE);	
				IF mcAxGdisable.Done THEN
					baxGenable := FALSE;
					MC.axGexecuteToFalse();
					iState := iState + 10;
				END_IF
			ELSE
				iState := iState + 10;
			END_IF	
			
	110:	// Homing
		io.fbXlhMotionAxisX.bHoming := TRUE;
		io.fbXlhMotionAxisX.fVelHoming := fVEL_HOMING;
		io.fbXlhMotionAxisX.fVelHomingFast := 3.0 * fVEL_HOMING;
		io.fbXlhMotionAxisX.eMcHomingDirection := MC_DIRECTION.positive;
		io.fbXlhMotionAxisX.fOffset := -168.5;
		
		io.fbXlhMotionAxisY.bHoming := TRUE;
		io.fbXlhMotionAxisY.fVelHoming := fVEL_HOMING;
		io.fbXlhMotionAxisY.fVelHomingFast := 3.0 * fVEL_HOMING;
		io.fbXlhMotionAxisY.eMcHomingDirection := MC_DIRECTION.positive;
		io.fbXlhMotionAxisY.fOffset := -31.0;
		
		io.fbXlhMotionAxisZ.bHoming := TRUE;
		io.fbXlhMotionAxisZ.fVelHoming := fVEL_HOMING;
		io.fbXlhMotionAxisZ.fVelHomingFast := 3.0 * fVEL_HOMING;
		io.fbXlhMotionAxisZ.eMcHomingDirection := MC_DIRECTION.positive;
		io.fbXlhMotionAxisZ.fOffset := -18.0;
		
		io.fbXlhMotionAxisA.bHoming := TRUE;
		io.fbXlhMotionAxisA.fVelHoming := fVEL_HOMING;
		//io.fbXlhMotionAxisA.rVelHomingFast := 3.0 * VEL_HOMING;
		io.fbXlhMotionAxisA.eMcHomingDirection := MC_DIRECTION.positive;
		//io.fbXlhMotionAxisA.rOffset := 0.0;
		
		IF io.fbXlhMotionAxisX.bHomingDone AND
			io.fbXlhMotionAxisY.bHomingDone AND
			io.fbXlhMotionAxisZ.bHomingDone AND
			io.fbXlhMotionAxisA.bHomingDone THEN
			axSmExecuteToFalse();
			io.fbXlhMotionAxisX.bHoming := FALSE;
			io.fbXlhMotionAxisY.bHoming := FALSE;
			io.fbXlhMotionAxisZ.bHoming := FALSE;
			io.fbXlhMotionAxisA.bHoming := FALSE;
			iState := iState + 10;
		END_IF	

	120:	// Enable der Achsengruppe
			IF NOT baxGenable THEN 
				mcAxGenable(AxisGroup := AxisGroup, Execute := TRUE);	
				IF mcAxGenable.Done THEN
					baxGenable := TRUE;
					MC.axGexecuteToFalse();
					iState := iState + 10;
					//iState := 580;
				END_IF			
			ELSE
				iState := iState + 10;
				//iState := 580;
			END_IF

	130: 	axSmExecuteToFalse();
			axGexecuteToFalse();	
			fbPickAndPlace.bExecute := FALSE;
			iState := iState + 10;		

	140: 
 		iState := 1000;

	// ============================================================================================
	// Kommandos
	// ============================================================================================
	
	1000: 	// Resetierung der Kommandos
		axX.fVel := fVEL;
		axX.fAcc := fACC_DEC;
		axX.fJerk := fJERK;
		
		axY.fVel := fVEL;
		axY.fAcc := fACC_DEC;
		axY.fJerk := fJERK;
		
		axZ.fVel := fVEL;
		axZ.fAcc := fACC_DEC;
		axZ.fJerk := fJERK;
		
		MC.axSmExecuteToFalse();
		MC.axGexecuteToFalse();		
		iState := iState + 10;
		
	1010:	// warte auf Aktion		
		//IF io.gpio.bSw5 THEN iState := 2000; END_IF
		//IF io.gpio.bSw6 THEN iState := 2010; END_IF
		//IF io.gpio.bSw5 THEN iState := 2020; END_IF
		//IF io.gpio.bSw6 THEN iState := 2030; END_IF
		//IF io.gpio.bSw5 THEN iState := 2040; END_IF
		//IF io.gpio.bSw6 THEN iState := 2050; END_IF
		//IF io.gpio.bSw5 THEN iState := 2060; END_IF
		//IF io.gpio.bSw6 THEN iState := 2070; END_IF
		//iState := 3000;
		//iState := 4000;
		
		
		IF bXp THEN smcPosRef.c.X := fStep;      smcPosRef.c.Y := 0.0;	      smcPosRef.c.Z := 0.0;        iState := 2000; END_IF
		IF bXm THEN smcPosRef.c.X := fStep*(-1); smcPosRef.c.Y := 0.0;	      smcPosRef.c.Z := 0.0;        iState := 2000; END_IF
		IF bYp THEN smcPosRef.c.X := 0.0;        smcPosRef.c.Y := fStep;	  smcPosRef.c.Z := 0.0;        iState := 2000; END_IF
		IF bYm THEN smcPosRef.c.X := 0.0;        smcPosRef.c.Y := fStep*(-1); smcPosRef.c.Z := 0.0;        iState := 2000; END_IF
		IF bZp THEN smcPosRef.c.X := 0.0;        smcPosRef.c.Y := 0.0;	      smcPosRef.c.Z := fStep;      iState := 2000; END_IF
		IF bZm THEN smcPosRef.c.X := 0.0;        smcPosRef.c.Y := 0.0;	      smcPosRef.c.Z := fStep*(-1); iState := 2000; END_IF
		IF bAuto THEN iState := 3000; END_IF


	// ============================================================================================
	// Stepbetrieb der Achsen
	// ============================================================================================
	
	2000: 	// relative Bewegung

			fbAxGmr.bExecute := TRUE;
			fbAxGmr.tPosRef := smcPosRef;
			IF fbAxGmr.bDone THEN
				MC.axGexecuteToFalse();
				iState := 1000;
			END_IF
			
	2010: 	// absolute Bewegung
			fbAxGma.bExecute := TRUE;
			fbAxGma.tPosRef := smcPosRef;
			IF fbAxGma.bDone THEN
				MC.axGexecuteToFalse();
				iState := 1000;
			END_IF

	// ============================================================================================
	// Pick and Place
	// ============================================================================================

	3000:	
			iI := 0;
			iN := 0;
			iState := iState + 10;	
				
	3010:	
			CASE iN OF
				0:
					fPickOffsetX :=     0.0;
					fPickOffsetY :=     0.0;
					fPlaceOffsetX :=   20.0;		
					fPlaceOffsetY :=   20.0;		
				1: 
					fPickOffsetX :=    20.0;
					fPickOffsetY :=    20.0;
					fPlaceOffsetX :=   20.0;		
					fPlaceOffsetY :=  -20.0;	
				2:
					fPickOffsetX :=    20.0;
					fPickOffsetY :=   -20.0;
					fPlaceOffsetX :=  -20.0;		
					fPlaceOffsetY :=  -20.0;			
				3: 
					fPickOffsetX :=   -20.0;
					fPickOffsetY :=   -20.0;
					fPlaceOffsetX :=  -20.0;		
					fPlaceOffsetY :=   20.0;
				4: 
					fPickOffsetX :=   -20.0;
					fPickOffsetY :=    20.0;
					fPlaceOffsetX :=   0.0;		
					fPlaceOffsetY :=   0.0;	
			END_CASE
			iState := iState + 10;	
	
	3020:
			CASE iI OF
				0:
					fOffsetX :=   0.0;
					fOffsetY :=   0.0;				
				1: 
					fOffsetX :=  70.0;
					fOffsetY :=   0.0;		
				2:
					fOffsetX :=  70.0;
					fOffsetY := -70.0;				
				3: 
					fOffsetX :=   0.0;
					fOffsetY := -70.0;		
			END_CASE
			iState := iState + 10;	

	3030: 	
			fbPickAndPlace.tPosPick.c.X := POS_REF.c.X + fPickOffsetX + fOffsetX;
			fbPickAndPlace.tPosPick.c.Y := POS_REF.c.Y + fPickOffsetY + fOffsetY;
			fbPickAndPlace.tPosPick.c.Z := POS_REF.c.Z;
			fbPickAndPlace.tPosPlace.c.X := POS_REF.c.X + fPlaceOffsetX + fOffsetX;
			fbPickAndPlace.tPosPlace.c.Y := POS_REF.c.Y + fPlaceOffsetY + fOffsetY;
			fbPickAndPlace.tPosPlace.c.Z := POS_REF.c.Z;
			fbPickAndPlace.bExecute := TRUE;
			io.bMagnet := fbPickAndPlace.bMagnet;
			IF fbPickAndPlace.bDone THEN
				fbPickAndPlace.bExecute := FALSE;
				axGexecuteToFalse();
				iState := iState + 10;
			END_IF
					
	3040:	
			iI := iI + 1;
			IF iI > 3 THEN
				iI := 0;
				iState := iState + 10;
			ELSE
				iState := 3020;
			END_IF
				
			
	3050:	
			iN := iN + 1;
			IF iN > 4 THEN
				iN := 0;
				iState := iState + 10;
			ELSE
				iState := 3010;
			END_IF
			
	3060:	IF bAuto THEN
				iState := 3000;
			ELSE
				iState := 1000;
			END_IF	
	
END_CASE

fbTonDelay1();
fbTonDelay2();
fbTonDelay1.IN := FALSE;
fbTonDelay2.IN := FALSE;

MC.write();

ACTION write:
io.write();
END_ACTION

ACTION read:
io.read();
END_ACTION

ACTION axSmExecuteToFalse:
axX.executeToFalse();
axY.executeToFalse();
axZ.executeToFalse();
axA.executeToFalse();
END_ACTION

ACTION axGexecuteToFalse:
mcAxGenable(AxisGroup := AxisGroup, Execute := FALSE);
mcAxGdisable(AxisGroup := AxisGroup, Execute := FALSE);
mcAxGreset(AxisGroup := AxisGroup, Execute := FALSE);
mcAxGsetCoord(AxisGroup := AxisGroup, Execute := FALSE);

fbAxGma.bExecute := FALSE;
fbAxGmr.bExecute := FALSE;
mcAxGmla(AxisGroup := AxisGroup, Execute := FALSE);
mcAxGmlr(AxisGroup := AxisGroup, Execute := FALSE);
END_ACTION

END_PROGRAM

// xLH_base/app/MOTION_BASE/FB_PLC_OPEN_AXIS
FUNCTION_BLOCK FB_PLC_OPEN_AXIS
VAR_INPUT	
	fVel: LREAL := 200.0;
	fAcc: LREAL := 750.0;
	fDec: LREAL := 750.0;
	fJerk: LREAL := 10000.0;
	
	mcrs: MC_ReadStatus := (Enable:=TRUE);
	mcrae: MC_ReadAxisError := (Enable:=TRUE);
	mcr: MC_Reset;
	smcrfbe: SMC_ReadFBError;
	mcp: MC_Power := (Enable:=FALSE, bRegulatorOn:=FALSE, bDriveStart:=FALSE);
	mcs: MC_Stop;
	mcma: MC_MoveAbsolute := (Velocity:=100.0, Acceleration:=1000.0, Deceleration:=1000.0, Jerk:=10000.0);
	mcmr: MC_MoveRelative := (Velocity:=100.0, Acceleration:=1000.0, Deceleration:=1000.0, Jerk:=10000.0);
	mcmv: MC_MoveVelocity := (Velocity:=100.0, Acceleration:=1000.0, Deceleration:=1000.0, Jerk:=10000.0, Direction:=-1);// 1 Positiv, -1 Negativ	
	
	pAxis: POINTER TO AXIS_REF_SM3; 
	// https://content.helpme-codesys.com/en/libs/SM3_Drive_PosControl/Current/AXIS_REF_POSCONTROL.html
	//axisPosControl: REFERENCE TO AXIS_REF_POSCONTROL;
END_VAR
VAR_OUTPUT	
	bError: BOOL;
	fActPos: LREAL;
	fActVel: LREAL;
	fActAcc: LREAL;
END_VAR
VAR
	bDummy: BOOL;
END_VAR

// Aufruf der PLC OPEN Motionbausteine
plcOpen();

// Fehlerauswertung
bError := mcs.Error OR mcmr.Error OR mcma.Error OR mcmv.Error;

// Zuweisung der Motion Control Istwerte
IF pAxis > 16#0 THEN
	fActPos := pAxis^.fActPosition;
	fActVel := pAxis^.fActVelocity;
	fActAcc := pAxis^.fActAcceleration;
END_IF

// axis.nAxisState = SMC_AXIS_STATE.standstill
// axis.nAxisState = SMC_AXIS_STATE.standstill

ACTION plcOpen:
IF pAxis > 16#0 THEN
	// Aufruf der PLC Open Motion Control Baustein
	mcrs(Axis:=pAxis^);// MC_ReadStatus https://help.codesys.com/search;version=3.5.17.0;term=MC_ReadStatus
	mcrae(Axis:=pAxis^);// MC_ReadAxisError https://help.codesys.com/webapp/ML6Svtks37sht2hVC_6YLIhf2ZY%2FMC_ReadAxisError;product=SM3_Basic;version=4.9.0.0
	mcr(Axis:=pAxis^);// MC_Reset https://help.codesys.com/webapp/xiNnxNPAb5nA4ocm6PFB_cHgUb4%2FMC_Reset;product=SM3_Basic;version=4.9.0.0
	smcrfbe(Axis:=pAxis^);// SMC_ReadFBError https://help.codesys.com/webapp/xUeuGLdUseEDKMLaPLQmdZO45P8%2FSMC_ReadFBError;product=SM3_Basic;version=4.9.0.0
	mcp(Axis:=pAxis^);// MC_Power https://help.codesys.com/webapp/xiNnxNPAb5nA4ocm6PFB_cHgUb4%2FMC_Power;product=SM3_Basic;version=4.9.0.0
	//mch(Axis:=pAxis^);// MC_Home https://content.helpme-codesys.com/en/libs/SM3_Basic/Current/SM3_Basic/POUs/Movement/MC_Home.html
	
	mcs.Deceleration := fDec;
	mcs.Jerk := fJerk;
	mcs(Axis:=pAxis^);// MC_Stop https://help.codesys.com/webapp/xUeuGLdUseEDKMLaPLQmdZO45P8%2FSMC_ReadFBError;product=SM3_Basic;version=4.9.0.0
	
	mcma.Velocity := fVel;
	mcma.Acceleration := fVel;
	mcma.Deceleration := fDec;
	mcma.Jerk := fJerk;
	mcma(Axis:=pAxis^);// MC_MoveAbsolute https://help.codesys.com/webapp/74YgxSD47ycAkED81whSoB9i6wQ%2FMC_MoveAbsolute;product=SM3_Basic;version=4.9.0.0
	
	mcmr.Velocity := fVel;
	mcmr.Acceleration := fAcc;
	mcmr.Deceleration := fDec;
	mcmr.Jerk := fJerk;
	mcmr(Axis:=pAxis^);// MC_MoveRelative https://help.codesys.com/webapp/74YgxSD47ycAkED81whSoB9i6wQ%2FMC_MoveRelative;product=SM3_Basic;version=4.9.0.0
	
	mcmv.Velocity := fVel;
	mcmv.Acceleration := fAcc;
	mcmv.Deceleration := fDec;
	mcmv.Jerk := fJerk;
	mcmv(Axis:=pAxis^);// MC_MoveVelocity https://help.codesys.com/webapp/74YgxSD47ycAkED81whSoB9i6wQ%2FMC_MoveVelocity;product=SM3_Basic;version=4.9.0.0
	
	// SoftMotion: https://help.codesys.com/webapp/_sm_components;product=codesys_softmotion;version=4.10.0.0
	// Drive: https://help.codesys.com/webapp/_sm_inserting_connected_drive_devices;product=codesys_softmotion;version=4.10.0.0
	// SMC Error: https://help.codesys.com/webapp/4icXWiTEEU7jfvlz7ATrx-Bu-fs%2FSMC_ERROR;product=SM3_Basic;version=4.0.0.0
END_IF
END_ACTION

ACTION executeToFalse:
mcr.Execute := FALSE;
mcs.Execute := FALSE;
mcma.Execute := FALSE;
mcmr.Execute := FALSE;
mcmv.Execute := FALSE;

bDummy := mcrs.Error; 
bDummy := mcrae.Error;
bDummy := mcr.Error;
bDummy := mcp.Error;
bDummy := mcs.Error;
bDummy := mcma.Error;
bDummy := mcmr.Error;
bDummy := mcmv.Error;
END_ACTION

END_FUNCTION_BLOCK

// xLH_base/app/MOTION_BASE/FB_AXG_MOVE_RELATIVE
FUNCTION_BLOCK FB_AXG_MOVE_RELATIVE
VAR_INPUT
	bExecute: BOOL;
	tPosRef: SMC_POS_REF;
	axGmr: REFERENCE TO MC_MoveLinearRelative;
	axG: REFERENCE TO AXIS_GROUP_REF_SM3;
END_VAR
VAR_OUTPUT
	bDone: BOOL;
END_VAR

axGmr.Execute := bExecute;
axGmr.Distance := tPosRef;
axGmr.BufferMode := MC_BUFFER_MODE.BlendingHigh;
axGmr.TransitionMode := MC_TRANSITION_MODE.TMCornerDistance;
axGmr.TransitionParameter[0] := 50;
//axGmvTo.CoordSystem := SMC_COORD_SYSTEM.PCS_1;
axGmr.CoordSystem := SMC_COORD_SYSTEM.MCS;
bDone := axGmr.Done;

END_FUNCTION_BLOCK

// xLH_base/app/MOTION_BASE/FB_AXG_MOVE_ABSOLUTE
FUNCTION_BLOCK FB_AXG_MOVE_ABSOLUTE
VAR_INPUT
	bExecute: BOOL;
	tPosRef: SMC_POS_REF;
	axGma: REFERENCE TO MC_MoveLinearAbsolute;
	axG: REFERENCE TO AXIS_GROUP_REF_SM3;
END_VAR
VAR_OUTPUT
	bDone: BOOL;
END_VAR

axGma.Execute := bExecute;
axGma.Position := tPosRef;
axGma.BufferMode := MC_BUFFER_MODE.BlendingHigh;
axGma.TransitionMode := MC_TRANSITION_MODE.TMCornerDistance;
axGma.TransitionParameter[0] := 50;
//axGmvTo.CoordSystem := SMC_COORD_SYSTEM.PCS_1;
axGma.CoordSystem := SMC_COORD_SYSTEM.MCS;
bDone := axGma.Done;

END_FUNCTION_BLOCK

// xLH_base/app/MOTION_BASE/FB_AXG_PICK_AND_PLACE
FUNCTION_BLOCK FB_AXG_PICK_AND_PLACE
VAR_INPUT
	bExecute: BOOL;
	tPosPick: SMC_POS_REF;
	tPosPlace: SMC_POS_REF;
	fbAxGma: REFERENCE TO FB_AXG_MOVE_ABSOLUTE;
	fbAxGmr: REFERENCE TO FB_AXG_MOVE_RELATIVE;
END_VAR
VAR_OUTPUT
	iState: INT := 0;
	bDone: BOOL;
	bMagnet: BOOL;
END_VAR
VAR
	smcPosRef: SMC_POS_REF;
	tonDelay1: TON;
END_VAR
VAR CONSTANT
	OFFSET_Z: REAL := 10.0;
END_VAR

IF bExecute THEN
	CASE iState OF
		0:	iState := iState + 10;
			(*
			smcPosRef.c.X := 0.0; 
			smcPosRef.c.Y := 0.0; 
			smcPosRef.c.Z := 0.0;//((LREAL_TO_REAL(z_axis.fActPosition) + 4.0)*(-1.0));
			smcPosRef.c.A := 180.0;
			smcPosRef.c.B := 180.0;
			smcPosRef.c.C := 0.0;
			fbAxGmr.bExecute := TRUE;
			fbAxGmr.tPosRef := smcPosRef;
			IF fbAxGmr.bDone THEN
				MC.axGexecuteToFalse();
				iState := iState + 10;
			END_IF
			*)
		
		10:	
			smcPosRef.c.X := tPosPick.c.X; 
			smcPosRef.c.Y := tPosPick.c.Y; 
			smcPosRef.c.Z := tPosPick.c.Z + OFFSET_Z;
			//smcPosRef.c.A := 180.0;
			//smcPosRef.c.B := 180.0;
			//smcPosRef.c.C := 0.0;
			fbAxGma.bExecute := TRUE;
			fbAxGma.tPosRef := smcPosRef;
			IF fbAxGma.bDone THEN
				MC.axGexecuteToFalse();
				iState := iState + 10;
			END_IF
		
		20:	smcPosRef.c.X := tPosPick.c.X; 
			smcPosRef.c.Y := tPosPick.c.Y; 
			smcPosRef.c.Z := tPosPick.c.Z;
			//smcPosRef.c.A := 180.0;
			//smcPosRef.c.B := 180.0;
			//smcPosRef.c.C := 0.0;
			fbAxGma.bExecute := TRUE;
			fbAxGma.tPosRef := smcPosRef;
			IF fbAxGma.bDone THEN
				MC.axGexecuteToFalse();
				iState := iState + 10;
			END_IF
			
		30:	bMagnet := TRUE;
			tonDelay1.IN := TRUE;
			tonDelay1.PT := T#250MS;
			IF tonDelay1.Q THEN
				iState := iState + 10;
			END_IF
		
		40:	// PICK Z-Achse Neutral 
			smcPosRef.c.X := tPosPick.c.X; 
			smcPosRef.c.Y := tPosPick.c.Y; 
			smcPosRef.c.Z := tPosPick.c.Z + OFFSET_Z;
			//smcPosRef.c.A := 180.0;
			//smcPosRef.c.B := 180.0;
			//smcPosRef.c.C := 0.0;
			fbAxGma.bExecute := TRUE;
			fbAxGma.tPosRef := smcPosRef;
			IF fbAxGma.bDone THEN
				MC.axGexecuteToFalse();
				iState := iState + 10;
			END_IF
			
		50:	// PLACE Z-Achse Neutral 
			smcPosRef.c.X := tPosPlace.c.X; 
			smcPosRef.c.Y := tPosPlace.c.Y; 
			smcPosRef.c.Z := tPosPlace.c.Z + OFFSET_Z;
			//smcPosRef.c.A := 180.0;
			//smcPosRef.c.B := 180.0;
			//smcPosRef.c.C := 0.0;
			fbAxGma.bExecute := TRUE;
			fbAxGma.tPosRef := smcPosRef;
			IF fbAxGma.bDone THEN
				MC.axGexecuteToFalse();
				iState := iState + 10;
			END_IF
			
		60:	// PLACE 
			smcPosRef.c.X := tPosPlace.c.X; 
			smcPosRef.c.Y := tPosPlace.c.Y; 
			smcPosRef.c.Z := tPosPlace.c.Z;
			//smcPosRef.c.A := 180.0;
			//smcPosRef.c.B := 180.0;
			//smcPosRef.c.C := 0.0;
			fbAxGma.bExecute := TRUE;
			fbAxGma.tPosRef := smcPosRef;
			IF fbAxGma.bDone THEN
				MC.axGexecuteToFalse();
				iState := iState + 10;
			END_IF
			
		70:	bMagnet := FALSE;
			tonDelay1.IN := TRUE;
			tonDelay1.PT := T#250MS;
			IF tonDelay1.Q THEN
				iState := iState + 10;
			END_IF
			
		80:	// PLACE Z-Achse Neutral
			bMagnet := FALSE;
			smcPosRef.c.X := tPosPlace.c.X; 
			smcPosRef.c.Y := tPosPlace.c.Y; 
			smcPosRef.c.Z := tPosPlace.c.Z + OFFSET_Z;
			//smcPosRef.c.A := 180.0;
			//smcPosRef.c.B := 180.0;
			//smcPosRef.c.C := 0.0;
			fbAxGma.bExecute := TRUE;
			fbAxGma.tPosRef := smcPosRef;
			IF fbAxGma.bDone THEN
				MC.axGexecuteToFalse();
				iState := iState + 10;
			END_IF
			
		90: bDone := TRUE;
		
	END_CASE	
ELSE
	iState := 0;
	bMagnet := FALSE;
	bDone := FALSE;
END_IF

tonDelay1();
tonDelay1.IN := FALSE;

END_FUNCTION_BLOCK

// xLH_base/app/IO/FB_XLH_GPIO
FUNCTION_BLOCK FB_XLH_GPIO
VAR_INPUT
	bLed1: BOOL;
	bLed2: BOOL;
	bLed3: BOOL;
	bLed4: BOOL;
	bLed5: BOOL;
	bLed6: BOOL;
	bLed7: BOOL;	
END_VAR
VAR_OUTPUT
	bSw1: BOOL;
	bSw2: BOOL;
	bSw3: BOOL;
	bSw4: BOOL;
	bSw5: BOOL;
	bSw6: BOOL;
	bSw7: BOOL;
	bSw8: BOOL;
END_VAR

METHOD read : BOOL
VAR_INPUT
END_VAR
END_METHOD

METHOD write : BOOL
VAR_INPUT
END_VAR
END_METHOD

END_FUNCTION_BLOCK

// xLH_base/app/IO/FB_XLH_DXL_RGB
FUNCTION_BLOCK FB_XLH_DXL_RGB
VAR_INPUT
	uiDxl1PositionGet: UINT;
	iDxl1CurrentGet: INT;
	uiDxl2PositionGet: UINT;
	iDxl2CurrentGet: INT;

	bDxl1Torque: BOOL;
	bDxl1Led: BOOL;
	uiDxl1Position: UINT;
	uiDxl1Velocity: UINT;
	
	bDxl2Torque: BOOL;
	bDxl2Led: BOOL;
	uiDxl2Position: UINT;
	uiDxl2Velocity: UINT;
	
	byRgbRed: BYTE;
	byRgbGreen: BYTE;
	byRgbBlue: BYTE;
END_VAR
VAR_OUTPUT

END_VAR

METHOD read : BOOL
VAR_INPUT
END_VAR
END_METHOD

METHOD write : BOOL
VAR_INPUT
END_VAR
END_METHOD

END_FUNCTION_BLOCK

// xLH_base/app/IO/FB_XLH_MOTION
FUNCTION_BLOCK FB_XLH_MOTION
VAR_INPUT
	adiPosition: ARRAY[1..4] OF DINT;
	{attribute 'displaymode':='bin'} 
	abyInputs: ARRAY[1..3] OF BYTE;
	bAxXsw: BOOL;
	bAxYsw: BOOL;
	bAxZsw: BOOL;
	bSensor: BOOL;
	
	{attribute 'displaymode':='bin'} 
	abyControl: ARRAY[1..4] OF BYTE;
	afFrequencyCalc: ARRAY[1..4] OF LREAL;
	afbFilterFrequency: ARRAY[1..4] OF FB_KALMAN_FILTER;
	adiFrequency: ARRAY[1..4] OF DINT;
	uiMagnetDutyCycle: UINT;
	abyOutputs: ARRAY[1..2] OF BYTE;
	ausServo: ARRAY[1..8] OF USINT;
	
	pfbXlhMotionAxis: ARRAY [1..4] OF POINTER TO FB_XLH_MOTION_AXIS_BASE;
END_VAR
VAR_OUTPUT

END_VAR

METHOD read : BOOL
VAR_INPUT
END_VAR

(*
axX();
axY();
axZ();
axA();
fbXlhMotionAxisX();
fbXlhMotionAxisY();
fbXlhMotionAxisZ();
fbXlhMotionAxisA();
*)
pfbXlhMotionAxis[1]^.pfbAxisPlcOpen^();
pfbXlhMotionAxis[1]^();
pfbXlhMotionAxis[1]^.diPosition := adiPosition[1];
pfbXlhMotionAxis[1]^.mRead();

pfbXlhMotionAxis[2]^.pfbAxisPlcOpen^();
pfbXlhMotionAxis[2]^();
pfbXlhMotionAxis[2]^.diPosition := adiPosition[2];
pfbXlhMotionAxis[2]^.mRead();

pfbXlhMotionAxis[3]^.pfbAxisPlcOpen^();
pfbXlhMotionAxis[3]^();
pfbXlhMotionAxis[3]^.diPosition := adiPosition[3];
pfbXlhMotionAxis[3]^.mRead();

pfbXlhMotionAxis[4]^.pfbAxisPlcOpen^();
pfbXlhMotionAxis[4]^();
pfbXlhMotionAxis[4]^.diPosition := adiPosition[4];
pfbXlhMotionAxis[4]^.mRead();
END_METHOD

METHOD write : BOOL
VAR_INPUT
END_VAR
pfbXlhMotionAxis[1]^.mWrite();
pfbXlhMotionAxis[2]^.mWrite();
pfbXlhMotionAxis[3]^.mWrite();
pfbXlhMotionAxis[4]^.mWrite();

abyControl[1] := MEM.PackBitsToByte(
		FALSE,
		FALSE,
		pfbXlhMotionAxis[1]^.bMoveWithoutPulse,
		pfbXlhMotionAxis[1]^._bInMotion,
		pfbXlhMotionAxis[1]^.bInverted,
		pfbXlhMotionAxis[1]^.bReset,
		pfbXlhMotionAxis[1]^._bDir,
		pfbXlhMotionAxis[1]^._bEn);
afFrequencyCalc[1] := 150000000.0 / LIMIT(0.25, TO_REAL(pfbXlhMotionAxis[1]^._diFrequency), 50000.0);
afbFilterFrequency[1](fX:=afFrequencyCalc[1], fR:=1.0, fQ:=1.0);
adiFrequency[1] := LREAL_TO_DINT(LIMIT(2000.0, afbFilterFrequency[1].fY, 600000000.0));

abyControl[2] := MEM.PackBitsToByte(
		FALSE,
		FALSE,
		pfbXlhMotionAxis[2]^.bMoveWithoutPulse,
		pfbXlhMotionAxis[2]^._bInMotion,
		pfbXlhMotionAxis[2]^.bInverted,
		pfbXlhMotionAxis[2]^.bReset,
		pfbXlhMotionAxis[2]^._bDir,
		pfbXlhMotionAxis[2]^._bEn);
afFrequencyCalc[2] := 150000000.0 / LIMIT(0.25, TO_REAL(pfbXlhMotionAxis[2]^._diFrequency), 50000.0);
afbFilterFrequency[2](fX:=afFrequencyCalc[2], fR:=1.0, fQ:=1.0);
adiFrequency[2] := LREAL_TO_DINT(LIMIT(2000.0, afbFilterFrequency[2].fY, 600000000.0));

abyControl[3] := MEM.PackBitsToByte(
		FALSE,
		FALSE,
		pfbXlhMotionAxis[3]^.bMoveWithoutPulse,
		pfbXlhMotionAxis[3]^._bInMotion,
		pfbXlhMotionAxis[3]^.bInverted,
		pfbXlhMotionAxis[3]^.bReset,
		pfbXlhMotionAxis[3]^._bDir,
		pfbXlhMotionAxis[3]^._bEn);
afFrequencyCalc[3] := 150000000.0 / LIMIT(0.25, TO_REAL(pfbXlhMotionAxis[3]^._diFrequency), 50000.0);
afbFilterFrequency[3](fX:=afFrequencyCalc[3], fR:=1.0, fQ:=1.0);
adiFrequency[3] := LREAL_TO_DINT(LIMIT(2000.0, afbFilterFrequency[3].fY, 600000000.0));

abyControl[4] := MEM.PackBitsToByte(
		FALSE,
		FALSE,
		pfbXlhMotionAxis[4]^.bMoveWithoutPulse,
		pfbXlhMotionAxis[4]^._bInMotion,
		pfbXlhMotionAxis[4]^.bInverted,
		pfbXlhMotionAxis[4]^.bReset,
		pfbXlhMotionAxis[4]^._bDir,
		pfbXlhMotionAxis[4]^._bEn);
afFrequencyCalc[4] := 150000000.0 / LIMIT(0.25, TO_REAL(pfbXlhMotionAxis[4]^._diFrequency), 50000.0);
afbFilterFrequency[4](fX:=afFrequencyCalc[4], fR:=1.0, fQ:=1.0);
adiFrequency[4] := LREAL_TO_DINT(LIMIT(2000.0, afbFilterFrequency[4].fY, 600000000.0));
END_METHOD

END_FUNCTION_BLOCK

// xLH_base/app/MOTION_BASE/FB_KALMAN_FILTER
FUNCTION_BLOCK PUBLIC FB_KALMAN_FILTER
VAR_INPUT
	fX: LREAL;
	fQ: LREAL;
	fR: LREAL;
	bReset: BOOL;
END_VAR
VAR_OUTPUT
	fY: LREAL;
END_VAR
VAR 
	X_hat: LREAL;
	X_hat_min: LREAL;
	poise: LREAL;
	Pmin: LREAL;
	K: LREAL;
	fAvoidZero: LREAL := 0.001;
END_VAR

IF bReset THEN
	reset();
END_IF

K := Pmin/MAX((Pmin + fR), fAvoidZero);
X_hat := X_hat_min + K*(fX - X_hat_min);
poise := (1 - K)*Pmin;
Pmin := poise + fQ;
X_hat_min := X_hat;
fY := X_hat;

ACTION reset:
X_hat := 0.0;
X_hat_min := 0.0;
poise := 0.0;
Pmin := 0.0;
K := 0.0;
fY := 0.0;
END_ACTION

END_FUNCTION_BLOCK

// xLH_base/app/MOTION_BASE/FB_XLH_MOTION_AXIS_BASE
FUNCTION_BLOCK FB_XLH_MOTION_AXIS_BASE
VAR_INPUT
	bInverted: BOOL;
	bReset: BOOL;
	bMoveWithoutPulse: BOOL;
	diPosition: DINT;
	pAxis: POINTER TO AXIS_REF_POSCONTROL;
	pfbAxisPlcOpen: POINTER TO FB_PLC_OPEN_AXIS;
END_VAR
VAR_OUTPUT
	
END_VAR
VAR
	_fbTofSm1: TOF;
	_bEn: BOOL;
	_bDir: BOOL;
	_bInMotion: BOOL;
	_diFrequency: DINT;	
END_VAR

METHOD mRead : BOOL
VAR_INPUT
END_VAR
VAR

END_VAR
IF pAxis > 16#0 THEN
	pAxis^.in.dwActPosition := TO_DWORD(diPosition);
	pAxis^.in.bDriveStartRealState := TRUE;
	pAxis^.in.bRegulatorRealState := TRUE;
END_IF
END_METHOD

METHOD mWrite : BOOL
VAR_INPUT
END_VAR
VAR

END_VAR
IF pAxis > 16#0 THEN
	_bDir := (pAxis^.out.diSetVelocity >= 0);
	_diFrequency := ABS(pAxis^.out.diSetVelocity);
	// https://content.helpme-codesys.com/en/libs/SM3_Basic/Current/SM3_Basic/DataTypes/DriveInterface/SMC_AXIS_STATE.html
	_bEn := (pAxis^.nAxisState >= 1);
	_fbTofSm1(IN:=(pAxis^.nAxisState >= 4), PT:=T#500MS, Q=>_bInMotion);
END_IF
END_METHOD

END_FUNCTION_BLOCK

// xLH_base/app/MOTION_BASE/FB_XLH_MOTION_AXIS_SIMPLE_ES
FUNCTION_BLOCK FB_XLH_MOTION_AXIS_SIMPLE_ES EXTENDS FB_XLH_MOTION_AXIS_BASE
VAR_INPUT
	bHoming: BOOL;
	fVelHoming: LREAL;
	fVelHomingFast: LREAL;
	eMcHomingDirection: MC_Direction;
	fOffset: LREAL;
	pbEs: POINTER TO BOOL;
END_VAR
VAR_OUTPUT
	bHomingDone: BOOL;
	bEs: BOOL;
END_VAR
VAR
	iState: INT;
	fbTonDelay1: TON;
END_VAR
VAR CONSTANT
	rOFFSET_HOMING: real := 3.0;
END_VAR

SUPER^();
bReset := FALSE; 
bMoveWithoutPulse := FALSE; 
bHomingDone := FALSE;
IF NOT bHoming THEN
	iState := 0;
END_IF

IF pfbAxisPlcOpen > 16#0 THEN
	CASE iState OF
		0: 		IF bHoming THEN
					iState := 100;	
				END_IF
				
		100:	pfbAxisPlcOpen^.fVel := fVelHomingFast;
				pfbAxisPlcOpen^.mcmv.Execute := TRUE;
				pfbAxisPlcOpen^.mcmv.Direction := eMcHomingDirection;
				IF NOT bEs THEN
					pfbAxisPlcOpen^.executeToFalse();
					iState := iState + 10;
				END_IF
				
		110:	pfbAxisPlcOpen^.mcs.Execute := TRUE;
				IF pfbAxisPlcOpen^.mcs.Done THEN
					pfbAxisPlcOpen^.executeToFalse();
					iState := iState + 10;
				END_IF
				
				
		120:	pfbAxisPlcOpen^.mcmr.Execute := TRUE;
				pfbAxisPlcOpen^.fVel := fVelHoming;
				IF eMcHomingDirection = MC_DIRECTION.negative THEN
					pfbAxisPlcOpen^.mcmr.Distance := rOFFSET_HOMING;
				ELSE
					pfbAxisPlcOpen^.mcmr.Distance := (-1.0) * rOFFSET_HOMING;
				END_IF
				IF pfbAxisPlcOpen^.mcmr.Done THEN
					pfbAxisPlcOpen^.executeToFalse();
					iState := iState + 10;
				END_IF
				
		130:	pfbAxisPlcOpen^.fVel := fVelHoming;
				pfbAxisPlcOpen^.mcmv.Execute := TRUE;
				pfbAxisPlcOpen^.mcmv.Direction := eMcHomingDirection;
				IF NOT bEs THEN
					pfbAxisPlcOpen^.executeToFalse();
					iState := iState + 10;
				END_IF
				
		140:	pfbAxisPlcOpen^.mcs.Execute := TRUE;
				IF pfbAxisPlcOpen^.mcs.Done THEN
					pfbAxisPlcOpen^.executeToFalse();
					iState := iState + 10;
				END_IF		
				
		150:	pfbAxisPlcOpen^.mcmr.Execute := TRUE;
				pfbAxisPlcOpen^.fVel := TO_REAL(pfbAxisPlcOpen^.pAxis^.fSWMaxVelocity); 
				pfbAxisPlcOpen^.mcmr.Distance := fOffset;
				IF pfbAxisPlcOpen^.mcmr.Done THEN
					pfbAxisPlcOpen^.executeToFalse();
					iState := iState + 10;
				END_IF
				
		160:	//bReset := TRUE; 
				bMoveWithoutPulse := TRUE; 
				pfbAxisPlcOpen^.mcma.Execute := TRUE;
				pfbAxisPlcOpen^.fVel := TO_REAL(pfbAxisPlcOpen^.pAxis^.fSWMaxVelocity); 
				pfbAxisPlcOpen^.mcma.Position := 0.0;
				IF pfbAxisPlcOpen^.mcma.Done THEN
					pfbAxisPlcOpen^.executeToFalse();
					iState := iState + 10;
				END_IF
				
		170:	//bReset := TRUE; 
				bMoveWithoutPulse := TRUE; 
				fbTonDelay1.IN := TRUE;
				fbTonDelay1.PT := T#250MS;
				IF fbTonDelay1.Q THEN
					iState := iState + 10;
				END_IF
		
		180: 	bHomingDone := TRUE;
		
		ELSE 	iState := 0;
	END_CASE
ELSE
	iState := 0;
END_IF

fbTonDelay1();
fbTonDelay1.IN := FALSE;

METHOD mRead : BOOL
VAR_INPUT
END_VAR
VAR

END_VAR
SUPER^.mRead();
IF pbEs > 16#0 THEN
	bEs := pbEs^;
ELSE
	bEs := FALSE;
END_IF
END_METHOD

END_FUNCTION_BLOCK

// xLH_base/app/MOTION_BASE/FB_XLH_MOTION_AXIS_SIMPLE
FUNCTION_BLOCK FB_XLH_MOTION_AXIS_SIMPLE EXTENDS FB_XLH_MOTION_AXIS_BASE
VAR_INPUT
	bHoming: BOOL;
	fVelHoming: LREAL;
	eMcHomingDirection: MC_Direction;
END_VAR
VAR_OUTPUT
	bHomingDone: BOOL;
END_VAR
VAR
	iState: INT;
	fbTonDelay1: TON;
END_VAR

SUPER^();
bReset := FALSE; 
bMoveWithoutPulse := FALSE; 
bHomingDone := FALSE;
IF NOT bHoming THEN
	iState := 0;
END_IF

IF pfbAxisPlcOpen > 16#0 THEN
	CASE iState OF
		0: 		IF bHoming THEN
					iState := 100;	
				END_IF
						
		100:	bReset := TRUE; 
				bMoveWithoutPulse := TRUE; 
				pfbAxisPlcOpen^.mcma.Execute := TRUE;
				pfbAxisPlcOpen^.fVel := fVelHoming * 10.0; 
				pfbAxisPlcOpen^.mcma.Position := 0.0;
				IF pfbAxisPlcOpen^.mcma.Done THEN
					pfbAxisPlcOpen^.executeToFalse();
					iState := iState + 10;
				END_IF
				
		110:	bReset := TRUE; 
				bMoveWithoutPulse := TRUE; 
				fbTonDelay1.IN := TRUE;
				fbTonDelay1.PT := T#100MS;
				IF fbTonDelay1.Q THEN
					bReset := FALSE; 
					bMoveWithoutPulse := FALSE;
					iState := iState + 10;
				END_IF
		
		120: 	bHomingDone := TRUE;
		
		ELSE 	iState := 0;
	END_CASE
ELSE
	iState := 0;
END_IF

fbTonDelay1();
fbTonDelay1.IN := FALSE;

END_FUNCTION_BLOCK

// xLH_base/app/MAIN_CALLER
PROGRAM MAIN_CALLER
VAR
	bDevicesCoRunning: BOOL;
	fbTonDevicesCoRunning: TON := (PT:=T#250MS);
END_VAR

// Ueberwachung ob alle CAN-Open Devices im Status RUN sind
(*
fbTonDevicesCoRunning(IN:= 
	(xlh_motion.CANopenState = _3SCOS.DEVICE_STATE.OPERATIONAL) AND
	(xlh_dynamixel_rgb.CANopenState = _3SCOS.DEVICE_STATE.OPERATIONAL)	
);
*)
fbTonDevicesCoRunning(IN:= 
	(xlh_motion.CANopenState = _3SCOS.DEVICE_STATE.OPERATIONAL)
);
// falls alle Devices im Status RUN sind (inklusive Verzögerung), wird die POE MAIN aufgerufen
IF fbTonDevicesCoRunning.Q THEN
	MC();
END_IF

END_PROGRAM

// xLH_base/app/Visualization
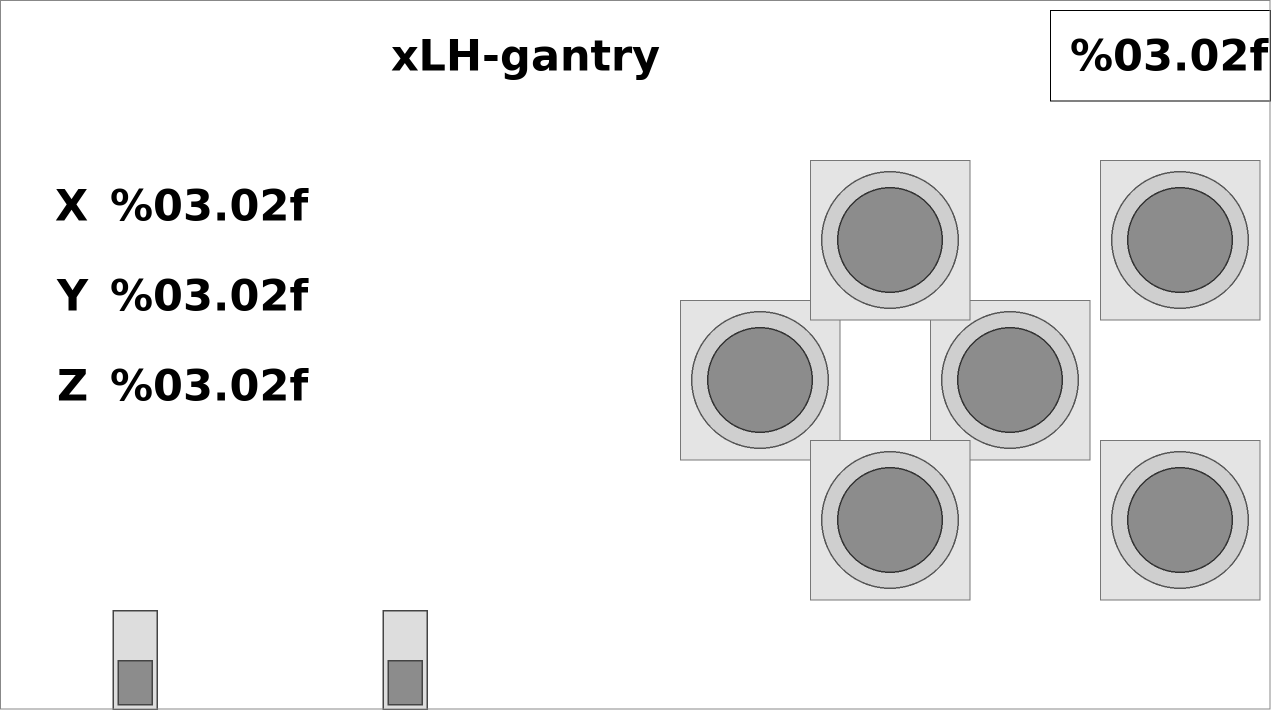
VISUALIZATION Visualization  // 1271x710
    PushSwitch (680,300 160x160), variable: MC.bXm, behaviour: TAP, style: Switch-PushSwitch-Gray
    PushSwitch (930,300 160x160), variable: MC.bXp, behaviour: TAP, style: Switch-PushSwitch-Gray
    PushSwitch (810,160 160x160), variable: MC.bYp, behaviour: TAP, style: Switch-PushSwitch-Gray
    PushSwitch (810,440 160x160), variable: MC.bYm, behaviour: TAP, style: Switch-PushSwitch-Gray
    PushSwitch (1100,160 160x160), variable: MC.bZp, behaviour: TAP, style: Switch-PushSwitch-Gray
    PushSwitch (1100,440 160x160), variable: MC.bZm, behaviour: TAP, style: Switch-PushSwitch-Gray
    Rectangle (90,160 221x91), "%03.02f", text variable: MC.axX.fActPos
    Rectangle (0,10 1051x91), "xLH-gantry"
    Rectangle (10,160 81x91), "X"
    Rectangle (90,250 221x91), "%03.02f", text variable: MC.axY.fActPos
    Rectangle (10,250 81x91), "Y"
    Rectangle (90,340 221x91), "%03.02f", text variable: MC.axZ.fActPos
    Rectangle (10,340 81x91), "Z"
    Rectangle (1050,10 221x91), "%03.02f", text variable: MC.fStep
        OnMouseClick: write the text variable via VisuDialogs.NumpadExtended, min 0.1, max 50.0
    DipSwitch (10,610 250x100), variable: io.bMagnet, behaviour: TOGGLE, style: Switch-DipSwitch-Gray
    DipSwitch (280,610 250x100), variable: MC.bAuto, behaviour: TOGGLE, style: Switch-DipSwitch-Gray
END_VISUALIZATION
